SUBAPPLICATION GetEndpointFromOrchestrationForm (* Get the IP:PORT/URI endpoint from an Orchestration Form *)
  (* Standard: 61499-2; Description: Copyright (c) 2018 fortiss GmbH This program and the accompanying materials are made available under the terms of the Eclipse Public License 2.0 which is available at https://www.eclipse.org/legal/epl-2.0/ SPDX-License-Identifier: EPL-2.0 *)
  (* Version 1.0, 2018-09-21, Jose Cabral, fortiss GmbH *)
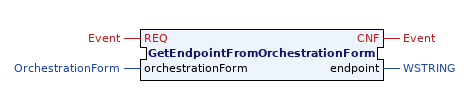
  EVENT_INPUT
    REQ; (* Request endpoint *)
  END_EVENT
  EVENT_OUTPUT
    CNF; (* Endpoint requested *)
  END_EVENT
  VAR_INPUT
    orchestrationForm : OrchestrationForm; (* Orchestration Form to look into *)
  END_VAR
  VAR_OUTPUT
    endpoint : WSTRING; (* Resulting endpoint from input *)
  END_VAR
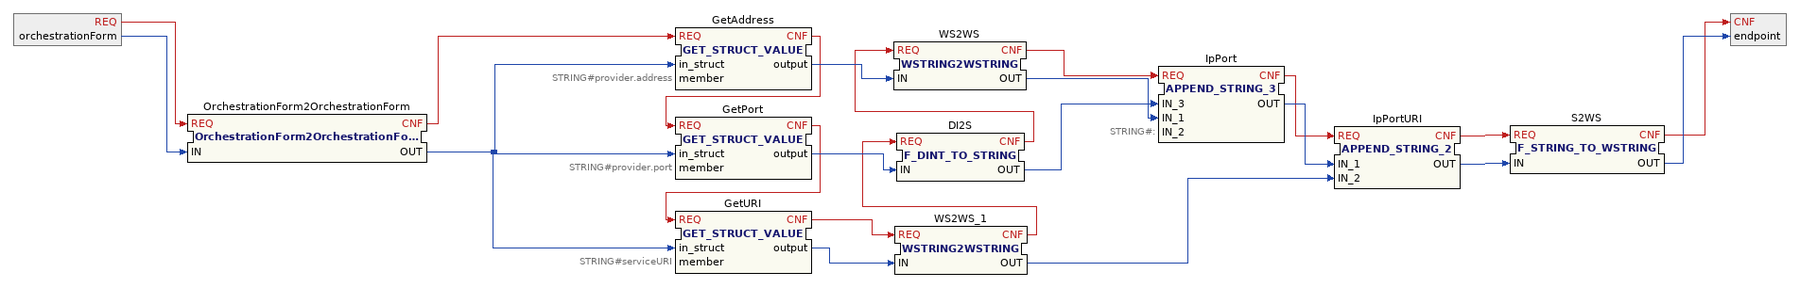
  FBS
    S2WS : F_STRING_TO_WSTRING;
    WS2WS : WSTRING2WSTRING;
    DI2S : F_DINT_TO_STRING;
    GetAddress : GET_STRUCT_VALUE(member := STRING#provider.address);
    GetPort : GET_STRUCT_VALUE(member := STRING#provider.port);
    GetURI : GET_STRUCT_VALUE(member := STRING#serviceURI);
    IpPort : APPEND_STRING_3(IN_2 := STRING#:);
    OrchestrationForm2OrchestrationForm : OrchestrationForm2OrchestrationForm;
    WS2WS_1 : WSTRING2WSTRING;
    IpPortURI : APPEND_STRING_2;
  END_FBS
  EVENT_CONNECTIONS
    DI2S.CNF TO WS2WS.REQ;
    GetPort.CNF TO GetURI.REQ;
    WS2WS.CNF TO IpPort.REQ;
    GetAddress.CNF TO GetPort.REQ;
    S2WS.CNF TO CNF;
    OrchestrationForm2OrchestrationForm.CNF TO GetAddress.REQ;
    REQ TO OrchestrationForm2OrchestrationForm.REQ;
    GetURI.CNF TO WS2WS_1.REQ;
    WS2WS_1.CNF TO DI2S.REQ;
    IpPort.CNF TO IpPortURI.REQ;
    IpPortURI.CNF TO S2WS.REQ;
  END_CONNECTIONS
  DATA_CONNECTIONS
    DI2S.OUT TO IpPort.IN_3;
    WS2WS.OUT TO IpPort.IN_1;
    GetPort.output TO DI2S.IN;
    GetAddress.output TO WS2WS.IN;
    S2WS.OUT TO endpoint;
    OrchestrationForm2OrchestrationForm.OUT TO GetAddress.in_struct;
    OrchestrationForm2OrchestrationForm.OUT TO GetPort.in_struct;
    OrchestrationForm2OrchestrationForm.OUT TO GetURI.in_struct;
    orchestrationForm TO OrchestrationForm2OrchestrationForm.IN;
    GetURI.output TO WS2WS_1.IN;
    IpPort.OUT TO IpPortURI.IN_1;
    IpPortURI.OUT TO S2WS.IN;
    WS2WS_1.OUT TO IpPortURI.IN_2;
  END_CONNECTIONS
END_SUBAPPLICATION
